PROGRAM MAIN
VAR
	TimeForInterlockDelay: TIME := T#0.05S;
	ManualMode: BOOL;
	MotorSelection_1: MotorSelection;
	SelectedMotor: INT;
	temp: TIME;
	LowerLeftInterlock: TOF;
	LowerLeft: BOOL;
	LowerRightInterlock: TOF;
	LowerRight: BOOL;
END_VAR
VAR // added by the converter: edge detectors and wires of the graphical bodies
    _w1, _w2, _w3, _w4 : BOOL;
END_VAR

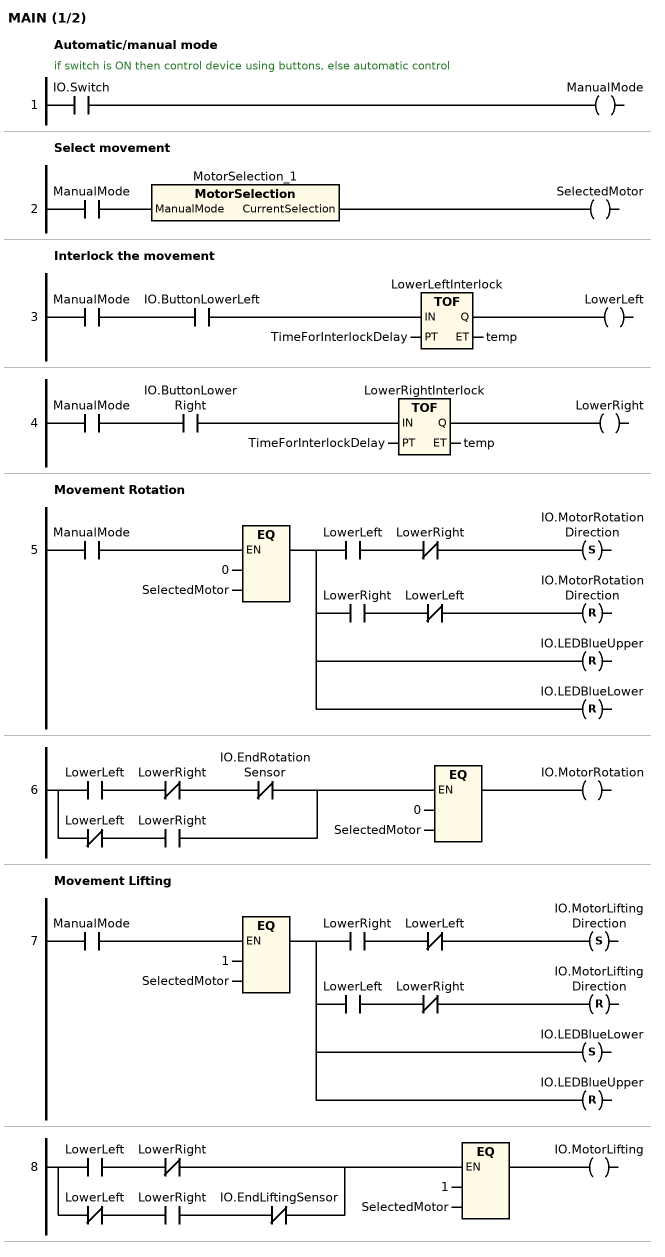
// NETWORK 1: Automatic/manual mode
// if switch is ON then control device using buttons, else automatic control
ManualMode := IO.Switch;

// NETWORK 2: Select movement
MotorSelection_1(ManualMode := ManualMode); // MotorSelection
SelectedMotor := MotorSelection_1.CurrentSelection;

// NETWORK 3: Interlock the movement
LowerLeftInterlock(IN := ManualMode AND IO.ButtonLowerLeft, PT := TimeForInterlockDelay, ET => temp); // TOF
LowerLeft := LowerLeftInterlock.Q;

// NETWORK 4
LowerRightInterlock(IN := ManualMode AND IO.ButtonLowerRight, PT := TimeForInterlockDelay, ET => temp); // TOF
LowerRight := LowerRightInterlock.Q;

// NETWORK 5: Movement Rotation
_w1 := ManualMode AND 0 = SelectedMotor;
IO.MotorRotationDirection S= _w1 AND LowerLeft AND NOT LowerRight;
IO.MotorRotationDirection R= _w1 AND LowerRight AND NOT LowerLeft;
IO.LEDBlueUpper R= _w1;
IO.LEDBlueLower R= _w1;

// NETWORK 6
IO.MotorRotation := (LowerLeft AND NOT LowerRight AND NOT IO.EndRotationSensor OR NOT LowerLeft AND LowerRight) AND 0 = SelectedMotor;

// NETWORK 7: Movement Lifting
_w2 := ManualMode AND 1 = SelectedMotor;
IO.MotorLiftingDirection S= _w2 AND LowerRight AND NOT LowerLeft;
IO.MotorLiftingDirection R= _w2 AND LowerLeft AND NOT LowerRight;
IO.LEDBlueLower S= _w2;
IO.LEDBlueUpper R= _w2;

// NETWORK 8
IO.MotorLifting := (LowerLeft AND NOT LowerRight OR NOT LowerLeft AND LowerRight AND NOT IO.EndLiftingSensor) AND 1 = SelectedMotor;

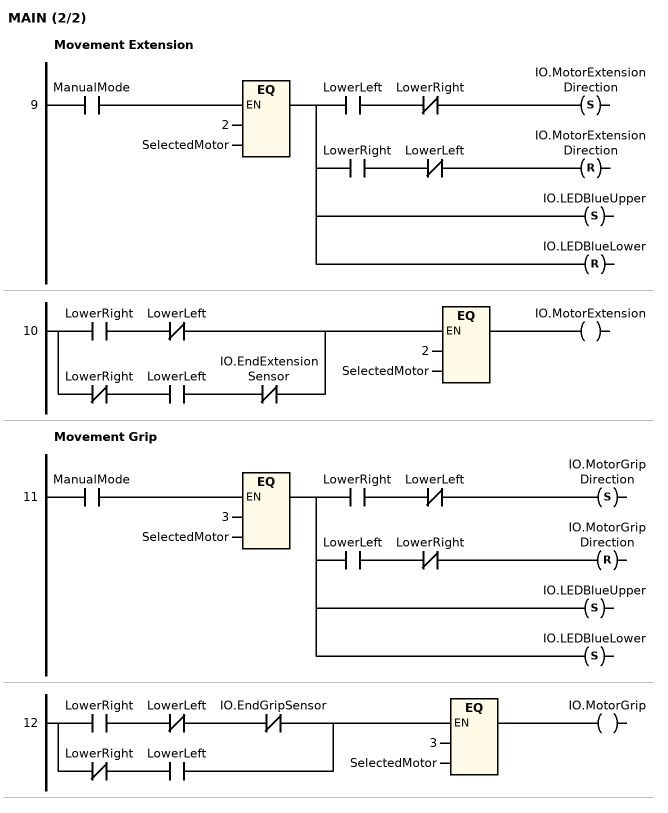
// NETWORK 9: Movement Extension
_w3 := ManualMode AND 2 = SelectedMotor;
IO.MotorExtensionDirection S= _w3 AND LowerLeft AND NOT LowerRight;
IO.MotorExtensionDirection R= _w3 AND LowerRight AND NOT LowerLeft;
IO.LEDBlueUpper S= _w3;
IO.LEDBlueLower R= _w3;

// NETWORK 10
IO.MotorExtension := (LowerRight AND NOT LowerLeft OR NOT LowerRight AND LowerLeft AND NOT IO.EndExtensionSensor) AND 2 = SelectedMotor;

// NETWORK 11: Movement Grip
_w4 := ManualMode AND 3 = SelectedMotor;
IO.MotorGripDirection S= _w4 AND LowerRight AND NOT LowerLeft;
IO.MotorGripDirection R= _w4 AND LowerLeft AND NOT LowerRight;
IO.LEDBlueUpper S= _w4;
IO.LEDBlueLower S= _w4;

// NETWORK 12
IO.MotorGrip := (LowerRight AND NOT LowerLeft AND NOT IO.EndGripSensor OR NOT LowerRight AND LowerLeft) AND 3 = SelectedMotor;

END_PROGRAM

(* stored: Version 1.1.0.1, ProductVersion 3.1.4024.13
   POU MAIN: Id {ca0d1193-1c86-427a-9c71-41bf6bccd822}, SpecialFunc None *)
